// SIMATIC S7-200 project (STEP 7-Micro/WIN), CPU 224XP REL 02.01

SYMBOL_TABLE USUARIO1
PMARCHA          I0.0
PARO             I0.1
TERMICO          I0.2
MOTOR            Q0.0
LEDMARCHA        Q0.1
LEDPARO          Q0.2
LEDDESCARGA      Q0.3
LEDAVERIA        Q0.4
RT               Q10.3
END_SYMBOL_TABLE

ORGANIZATION_BLOCK PRINCIPAL:OB1
TITLE=COMENTARIOS DEL PROGRAMA
BEGIN
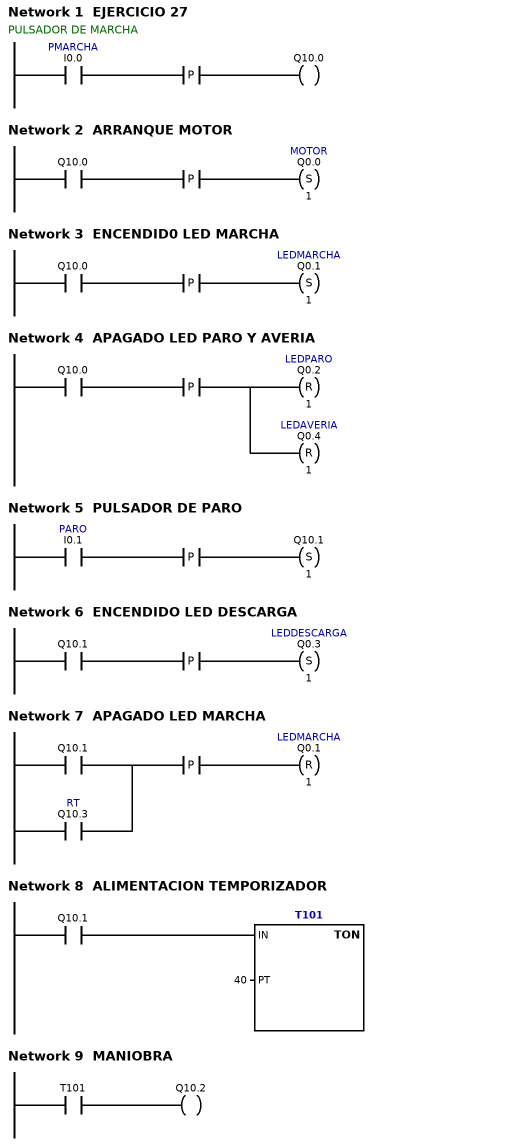
Network 1 // EJERCICIO 27
// PULSADOR DE MARCHA
LD     PMARCHA:I0.0
EU
=      Q10.0
Network 2 // ARRANQUE MOTOR
LD     Q10.0
EU
S      MOTOR:Q0.0, 1
Network 3 // ENCENDID0 LED MARCHA
LD     Q10.0
EU
S      LEDMARCHA:Q0.1, 1
Network 4 // APAGADO LED PARO Y AVERIA
LD     Q10.0
EU
R      LEDPARO:Q0.2, 1
R      LEDAVERIA:Q0.4, 1
Network 5 // PULSADOR DE PARO
LD     PARO:I0.1
EU
S      Q10.1, 1
Network 6 // ENCENDIDO LED DESCARGA
LD     Q10.1
EU
S      LEDDESCARGA:Q0.3, 1
Network 7 // APAGADO LED MARCHA
LD     Q10.1
O      RT:Q10.3
EU
R      LEDMARCHA:Q0.1, 1
Network 8 // ALIMENTACION TEMPORIZADOR
LD     Q10.1
TON    T101, 40
Network 9 // MANIOBRA
LD     T101
=      Q10.2
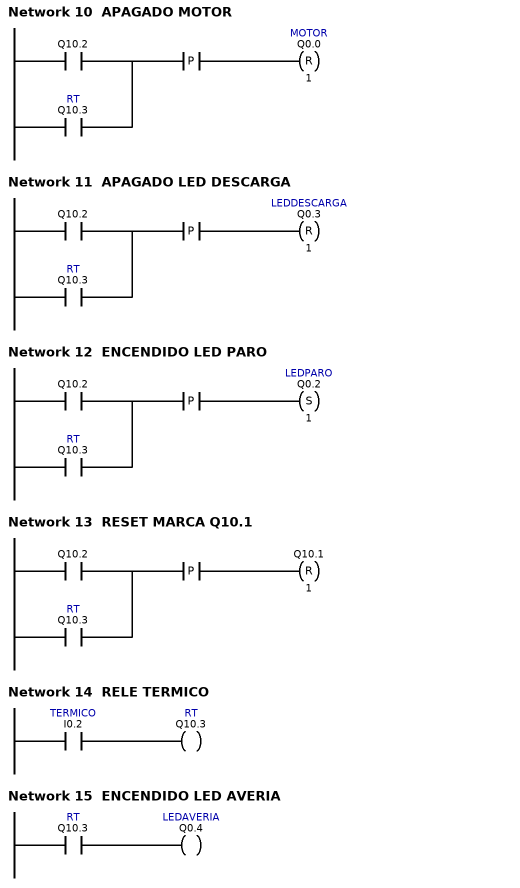
Network 10 // APAGADO MOTOR
LD     Q10.2
O      RT:Q10.3
EU
R      MOTOR:Q0.0, 1
Network 11 // APAGADO LED DESCARGA
LD     Q10.2
O      RT:Q10.3
EU
R      LEDDESCARGA:Q0.3, 1
Network 12 // ENCENDIDO LED PARO
LD     Q10.2
O      RT:Q10.3
EU
S      LEDPARO:Q0.2, 1
Network 13 // RESET MARCA Q10.1
LD     Q10.2
O      RT:Q10.3
EU
R      Q10.1, 1
Network 14 // RELE TERMICO
LD     TERMICO:I0.2
=      RT:Q10.3
Network 15 // ENCENDIDO LED AVERIA
LD     RT:Q10.3
=      LEDAVERIA:Q0.4
END_ORGANIZATION_BLOCK
